SUBAPPLICATION SIFB050 (* Subapplication Type *)
  (* Standard: 61499-2 *)
  (* Version 1.0, 2025-05-03, cochicde *)
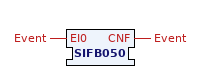
  EVENT_INPUT
    EI0;
  END_EVENT
  EVENT_OUTPUT
    CNF;
  END_EVENT
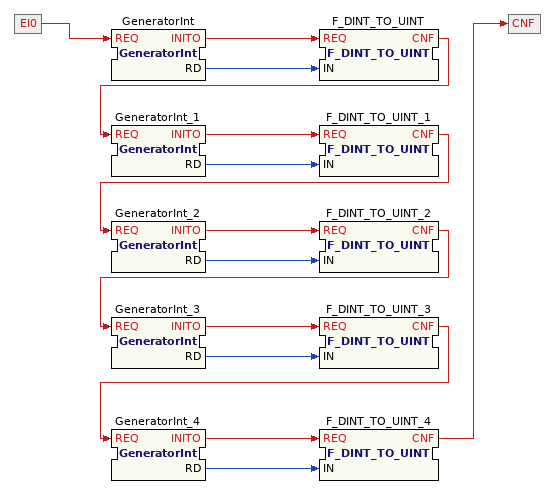
  FBS
    F_DINT_TO_UINT_1 : F_DINT_TO_UINT;
    F_DINT_TO_UINT_4 : F_DINT_TO_UINT;
    GeneratorInt : performance::GeneratorInt;
    GeneratorInt_2 : performance::GeneratorInt;
    GeneratorInt_1 : performance::GeneratorInt;
    F_DINT_TO_UINT_3 : F_DINT_TO_UINT;
    F_DINT_TO_UINT_2 : F_DINT_TO_UINT;
    GeneratorInt_4 : performance::GeneratorInt;
    F_DINT_TO_UINT : F_DINT_TO_UINT;
    GeneratorInt_3 : performance::GeneratorInt;
  END_FBS
  EVENT_CONNECTIONS
    GeneratorInt_1.INITO TO F_DINT_TO_UINT_1.REQ;
    F_DINT_TO_UINT_1.CNF TO GeneratorInt_2.REQ;
    GeneratorInt_4.INITO TO F_DINT_TO_UINT_4.REQ;
    GeneratorInt.INITO TO F_DINT_TO_UINT.REQ;
    GeneratorInt_2.INITO TO F_DINT_TO_UINT_2.REQ;
    F_DINT_TO_UINT.CNF TO GeneratorInt_1.REQ;
    GeneratorInt_3.INITO TO F_DINT_TO_UINT_3.REQ;
    F_DINT_TO_UINT_3.CNF TO GeneratorInt_4.REQ;
    F_DINT_TO_UINT_2.CNF TO GeneratorInt_3.REQ;
    EI0 TO GeneratorInt.REQ;
    F_DINT_TO_UINT_4.CNF TO CNF;
  END_CONNECTIONS
  DATA_CONNECTIONS
    GeneratorInt_1.RD TO F_DINT_TO_UINT_1.IN;
    GeneratorInt_4.RD TO F_DINT_TO_UINT_4.IN;
    GeneratorInt.RD TO F_DINT_TO_UINT.IN;
    GeneratorInt_2.RD TO F_DINT_TO_UINT_2.IN;
    GeneratorInt_3.RD TO F_DINT_TO_UINT_3.IN;
  END_CONNECTIONS
END_SUBAPPLICATION
